# EPICS substitutions: testIOC/testIOCApp/Db/user.substitutions
# Example substitutions file

file "db/circle.db" {
    { user = "jeonglee" }
}

file "db/dbExample1.db" {
    { user = "jeonglee" }
}

file db/dbExample2.db {
    pattern { user, no, scan }
        { "jeonglee", 1, "1 second" }
        { "jeonglee", 2, "2 second" }
        { "jeonglee", 3, "5 second" }
}
